{attribute 'linkalways'} 
{attribute 'no_explicit_call' := 'This FB is a CLASS and must be accessed using methods or properties'}
{attribute 'enable_dynamic_creation'}
FUNCTION_BLOCK Node_F_VN_MixImageChannels EXTENDS VisionNode
VAR
    ipSrcImage : _ITcVnImage;
    ipDestImage : _ITcVnImage;
    ipIndicesFromTo : _ITcVnContainer;
    hrPrev : _HRESULT(S_OK);
	hresult : _HRESULT(S_OK);
END_VAR

METHOD PUBLIC  Clone : I_Node
VAR
	pNode : POINTER TO Node_F_VN_MixImageChannels;
END_VAR
pNode := __NEW(Node_F_VN_MixImageChannels);
Clone := pNode^;
END_METHOD

METHOD FB_init : BOOL
VAR_INPUT
	bInitRetains : BOOL; // if TRUE, the retain variables are initialized (warm start / cold start)
	bInCopyCode : BOOL;  // if TRUE, the instance afterwards gets moved into the copy code (online change)
END_VAR
AddInput('ipSrcImage', ipSrcImage);
AddInput('ipIndicesFromTo', ipIndicesFromTo);
AddInput('hrPrev', hrPrev);
AddOutput('ipDestImage', ipDestImage);
AddOutput('hresult',hresult);
END_METHOD

METHOD PROTECTED OnExecute
hresult.Value := F_VN_MixImageChannels(
    ipSrcImage := ipSrcImage.Value,
	ipDestImage := ipDestImage.Value,
    ipIndicesFromTo := ipIndicesFromTo.Value,
	hrPrev := hrPrev.Value);
END_METHOD

METHOD PUBLIC PreExecutionCheck
VAR_INPUT
	Check : I_PreExecutionChecks;
END_VAR
Check.IsTrue(ipSrcImage.IsValid, 'ipSrcImage must contain an image');
Check.IsTrue(ipIndicesFromTo.IsType(TC_GLOBAL_CONST_LIST.ContainerType_Vector_TcVnVector2_DINT),
              'ipIndicesFromTo contains incorrect type');
END_METHOD

END_FUNCTION_BLOCK

(* stored: Version 1.1.0.1, ProductVersion 3.1.4026.13
   POU Node_F_VN_MixImageChannels: Id {1cb66c31-2d16-01da-1ddd-cc94fb119b8b}, SpecialFunc None
   Folder Constructor: Id {73c9bf1b-6077-09a3-3070-0c16197a133c}
   Method Clone: Id {58997106-d3dc-0b6b-189c-53d67df71bc5}
   Method FB_init: Id {b87d2220-ebf9-0106-2942-c14c4a44ceac}
   Method OnExecute: Id {c438ddc2-fecd-0c12-020e-4cecb9ec236c}
   Method PreExecutionCheck: Id {2cc7be21-01bb-086c-03a9-6590c0123e44} *)
